// TwinCAT 3 PLC project ModBus_Slave_PLC
// ProgramVersion: 3.1.4023.0
// libraries:
//   Tc2_ModbusSrv, * (Beckhoff Automation GmbH)
//   Tc2_Standard, * (Beckhoff Automation GmbH)
//   Tc2_System, * (Beckhoff Automation GmbH)
//   Tc3_Module, * (Beckhoff Automation GmbH)
// project tree:
//   GVLs/ GVL.TcGVL
//   / PlcTask.TcTTO
//   POUs/ MAIN.TcPOU
// real-time tasks:
//   TASK PlcTask: cycle T#10ms, priority 20, ADS port 350

CONFIGURATION ModBus_Slave_PLC
    RESOURCE PLC ON TwinCAT3
        TASK PlcTask(INTERVAL := T#10ms, PRIORITY := 20);
        PROGRAM MAIN WITH PlcTask : MAIN;
    END_RESOURCE
END_CONFIGURATION

// ---- GVLs/GVL.TcGVL
{attribute 'qualified_only'}
// These variable are mapped to the ModBus address ranges 0x8000 - 0x80FF for this device
VAR_GLOBAL
	mb_Input_Coils		: ARRAY[0..255] OF BOOL; // these coils can be queried by a MB master device using command 0x02
	mb_Output_Coils		: ARRAY[0..255] OF BOOL; // these coils can be set by a MB master device using 0x0f and queried by 0x01
	mb_Input_Registers	: ARRAY[0..255] OF WORD; // these registers are can be queried by a MB master device using command 0x04
	mb_Output_Registers	: ARRAY[0..255] OF WORD; // registers can be set by a MB device using 0x10, queried by 0x03 and 0x06
END_VAR

// ---- POUs/MAIN.TcPOU
PROGRAM MAIN
VAR
	bScroll			: BOOL;							// Set this to scroll the MB coils
	fbScrollTimer	: TON	:= (PT := T#0.1S);		// timer to scroll the MB registers  
	iIndex 			: INT;
	
	wPause	: WORD	:= 500;	// timer setting for scrolling MB coils 
	
END_VAR

// Set the modbus scroll if InputCoil 0 is set
IF(GVL.mb_Output_Coils[0] = TRUE) THEN
	bScroll	:= TRUE;
ELSE
	bScroll	:= FALSE;
END_IF

// get the pause time from Register 0
wPause				:= GVL.mb_Output_Registers[0];
fbScrollTimer.PT	:= WORD_TO_TIME(wPause);

// Scroll the ModBus coils if requested
IF(bScroll AND (wPause > 0)) THEN
	GVL.mb_Input_Coils[iIndex]	:= TRUE;
	fbScrollTimer(IN:=TRUE);		// run our send update timer  
	IF fbScrollTimer.Q THEN			// if the timer has expired (its time to set the registers) 
		fbScrollTimer(IN:=FALSE);  	// reset the timer 
		iIndex	:= iIndex + 1;	
		GVL.mb_Input_Coils[iIndex - 1]	:= FALSE;
		GVL.mb_Input_Coils[iIndex]		:= TRUE;
		IF(iIndex = 255) THEN
			iIndex	:= 0;
		END_IF
	END_IF	
END_IF

END_PROGRAM
